FUNCTION_BLOCK FB_Inmalen
VAR_INPUT

END_VAR
VAR_OUTPUT
END_VAR
VAR
		CurrentModus : E_Besturingsmodus := E_Besturingsmodus.uitlaten;
	KlepV2012 : ITF_OpenDichtKlep;
	KlepV2021 : ITF_OpenDichtKlep;
	KlepV2023 : ITF_OpenDichtKlep;
	KlepV2024 : ITF_OpenDichtKlep;
	
	SchuifV2013_AFG : ITF_Regelschuif;
	SchuifV2022_AFG : ITF_Regelschuif;
	
	SchuifV2013_DG : ITF_Regelschuif;
	SchuifV2022_DG : ITF_Regelschuif;
	
	pomp2_P2021 : ITF_Pomp;
	
	pompP2021 : INT;
END_VAR

CurrentModus:= main.Regelingen.BestuurMode;
IF CurrentModus = E_Besturingsmodus.inmalen THEN
	//set stand
	SchuifV2013_AFG.ActueelPosition := 0;
	SchuifV2013_DG.ActueelPosition := 0;	

	//set position
	KlepV2012.close();
	KlepV2021.Close();
	KlepV2024.Close();
	
	SchuifV2013_AFG.RegelSchuifGoTo(SchuifV2013_AFG.ActueelPosition);
	SchuifV2013_DG.RegelSchuifGoTo(SchuifV2013_DG.ActueelPosition);
	
	IF (KlepV2012.StateKlep = E_OpenDichtKlepState.closed AND
		KlepV2021.StateKlep = E_OpenDichtKlepState.closed AND
		KlepV2024.StateKlep = E_OpenDichtKlepState.closed AND
		SchuifV2013_AFG.StateRegelSchuif = E_RegelschuifState.standby AND
		SchuifV2013_DG.StateRegelSchuif = E_RegelschuifState.standby) THEN
		
		//set stand
		SchuifV2022_AFG.ActueelPosition := 100;
		SchuifV2022_DG.ActueelPosition := 100;
	
		//set position
		KlepV2023.Open();
		SchuifV2022_AFG.RegelSchuifGoTo(SchuifV2022_AFG.ActueelPosition);
		SchuifV2022_DG.RegelSchuifGoTo(SchuifV2022_DG.ActueelPosition);
		
		IF (KlepV2023.StateKlep = E_OpenDichtKlepState.open AND
			SchuifV2022_AFG.StateRegelSchuif = E_RegelschuifState.standby AND
			SchuifV2022_DG.StateRegelSchuif = E_RegelschuifState.standby) THEN
			
			//Get toerental
			pompP2021 := main.Regelingen.ToerentalP2021;
			
			//Set toerental
			pomp2_P2021.PompGoTo(pompP2021);
		END_IF	
	END_IF	
END_IF

METHOD FB_init : BOOL
VAR_INPUT
	bInitRetains : BOOL; // if TRUE, the retain variables are initialized (warm start / cold start)
	bInCopyCode : BOOL;  // if TRUE, the instance afterwards gets moved into the copy code (online change)
	OpenDichtKlepV2012 : ITF_OpenDichtKlep; 
	OpenDichtKlepV2021 : ITF_OpenDichtKlep; 
	OpenDichtKlepV2023 : ITF_OpenDichtKlep; 
	OpenDichtKlepV2024 : ITF_OpenDichtKlep; 
	
	RegelschuifV2013_AFO : ITF_Regelschuif; 
	RegelschuifV2022_AFO : ITF_Regelschuif;
	
	RegelschuifV2013_DG : ITF_Regelschuif;
	RegelschuifV2022_DG : ITF_Regelschuif;
	
	PompP2021 : ITF_Pomp;
	
END_VAR
KlepV2012 := OpenDichtKlepV2012;
KlepV2021 := OpenDichtKlepV2021;
KlepV2023 := OpenDichtKlepV2023;
KlepV2024 := OpenDichtKlepV2024;

SchuifV2013_AFG := RegelschuifV2013_AFO;
SchuifV2022_AFG := RegelschuifV2013_AFO;
SchuifV2013_DG := RegelschuifV2013_AFO;
SchuifV2022_DG := RegelschuifV2013_AFO;

pomp2_P2021 := PompP2021;
END_METHOD

END_FUNCTION_BLOCK

(* stored: Version 1.1.0.1, ProductVersion 3.1.4026.8
   POU FB_Inmalen: Id {96114e51-ad37-44de-ac67-1fd4ce3f2d17}, SpecialFunc None
   Method FB_init: Id {292cdf7f-9fce-4ac5-8a23-a71cd6cbd45e} *)
